// TIA Portal V21 export
DATA_BLOCK "SET VALUE"   // DB85
{ S7_Optimized_Access := 'FALSE' }
   VAR
      "PWD DOSING TIME" : String[80] := '  DOSING TIME (SEC)          :      60      ';
      "PWD WTR INLET TIME" : String[80] := '  WATER INLET TIME (MIN)     :       7     ';
      "PWD CRC TIME" : String[80] := '  CIRCULATION TIME (MIN)     :      10   ';
      "PWD DRAIN TIME" : String[80] := '  DRAIN TIME (MIN)           :       7    ';
      "STERILE TEMP1" : String[80] := '  HEAT UP-1 (DEG.C)          :    105.0  ';
      "STERILE TEMP2" : String[80] := '  HEAT UP-2 (DEG.C)          :    110.0  ';
      "STERILE TEMP3" : String[80] := '  HEAT UP-3 (DEG.C)          :    115.0  ';
      "STERILE TEMP4" : String[80] := '  STERILE TEMP (DEG.C)       :    121.4 ';
      "STERILE HOLD1" : String[80] := '  PULSE                      :       5    ';
      "STERILE HOLD2" : String[80] := '  PULSE                      :       5    ';
      "STERILE HOLD3" : String[80] := '  PULSE                      :       5    ';
      "STERILE HOLD4" : String[80] := '  HOLD TIME (MIN)            :      30    ';
      "WFI DSG TIME" : String[80] := '  DOSING TIME (SEC)          :      60 ';
      "WFI WTR TIME" : String[80] := '  WATER INLET TIME (MIN)     :       7 ';
      "WFI CRC TIME" : String[80] := '  CIRCULATION TIME (MIN)     :      10  ';
      "WFI DRAIN TIME" : String[80] := '  DRAIN TIME (MIN)           :      10  ';
      "STERILE EXH PRESS" : String[80] := '  EXHAUST PRESSURE (BAR)     :     0.05';
      "DRY VCC" : String[80] := '  VACUUM (BAR)               :    -0.500';
      "DRY VCC TIME" : String[80] := '  HOLD TIME (MIN)            :            ';
      "DRY ATS PRESSURE" : String[80] := '  ATMOSPHERIC PRESSURE (BAR) :    -0.050';
      "DRY TIME" : String[80] := '  DRYING TIME(MIN)           :      20     ';
      "PWD TEMP" : String[80] := '  PWD TEMP (DEG.C)           :     0.0    ';
      "STD TEMP1" : String[80] := '  HEAT UP-1 TEMPERATURE (DEG.C)         :   114.0       ';
      "STD TEMP2" : String[80] := '  HEAT UP-2 TEMPERATURE (DEG.C)         :   116.0       ';
      "STD TEMP3" : String[80] := '  HEAT UP-3 TEMPERATURE (DEG.C)         :   119.0       ';
      "STD TIME1" : String[80] := '  HEAT UP-1 HOLD TIME (MIN)             :      5     ';
      "STD TIME2" : String[80] := '  HEAT UP-2 HOLD TIME (MIN)             :      3     ';
      "STD TIME3" : String[80] := '  HEAT UP-3 HOLD TIME (MIN)             :      2     ';
      LEAK : String[80] := '  VACUUM (BAR)               :    -0.700';
      "DELAY BEFORE HOLD" : String[80] := '  DELAY BEFORE HOLD (MIN)    :       5';
      ACCEPTANCE : String[80] := '  ACCEPTANCE LEAKAGE (BAR)   :     0.013';
      "VCC HOLD" : String[80] := '  HOLD TIME (MIN)            :     10     ';
      "VCC PRESS" : String[80] := '  VENT PRESSURE (BAR)        :    -0.08';
      "HPHV VCC" : String[80] := '  PRE-VACUUM LEVEL (BAR)                :   -0.700      ';
      "HPHV VCC HOLD" : String[80] := '  PRE-VACUUM HOLD TIME (MIN)            :      3        ';
      "HPHV HEATUP" : String[80] := '  STERILIZATION TEMPERATURE (DEG.C)     :   121.4        ';
      "HPHV HEATUP HOLD" : String[80] := '  STERILIZATION HOLD TIME (MIN)         :     30       ';
      "HPHV NO" : String[80] := '  PRE-PULSE NUMBER                      :      3        ';
      "HPHV ATS" : String[80] := '  POST-VACUUM LEVEL (BAR)               :   -0.700      ';
      "HPHV ATS HOLD" : String[80] := '  POST-VACUUM HOLD TIME (MIN)           :     15        ';
      "HPHV EXH PRESS" : String[80] := '  EXHAUST PRESSURE (BAR)                :    0.2         ';
      "HPHV HEATUP PRESS" : String[80] := '  PRE-HEAT PRESSURE (BAR)               :    0.7        ';
      "HPHV END PRESS" : String[80] := '  END PRESSURE (BAR)                    :   -0.08       ';
      "BOW VCC" : String[80] := '  PRE-VACUUM LEVEL (BAR)                :   -0.700      ';
      "BOW VCC HOLD" : String[80] := '  PRE-VACUUM HOLD TIME (MIN)            :      3        ';
      "BOW HEATUP" : String[80] := '  STERILIZATION TEMPERATURE (DEG.C)     :   121.4        ';
      "BOW HEATUP HOLD" : String[80] := '  STERILIZATION HOLD TIME (MIN)         :     10       ';
      "BOW PRE PULSES" : String[80] := '  PRE-PULSE NUMBER                      :      3        ';
      "BOW POST VACUUM" : String[80] := '  POST-VACUUM LEVEL (BAR)               :    0.0        ';
      "BOW POST VACUUM HOLD" : String[80] := '  POST-VACUUM HOLD TIME (MIN)           :      0        ';   // 40:
      "BOW EXH PRESS" : String[80] := '  EXHAUST PRESSURE (BAR)                :    0.90        ';
      "BOW HEATUP PRESS" : String[80] := '  PRE-HEAT PRESSURE (BAR)               :    0.7        ';
      "BOW END PRESS" : String[80] := '  END PRESSURE (BAR)                    :    0.00       ';
      "STD UP PRESS" : String[80] := '  PRE PRESSURE (BAR)         :               0.00';
      "STD STOP TEMP" : String[80] := '  STERILIZATION STOP TEMP (DEG.C)       :   120.9     ';
      "STD VCC HOLD" : String[80] := '  VACUUM HOLD TIME (MIN)     :             ';
      "STD NO OF PULSES" : String[80] := '  NO OF PULSES               :                 0';
      "DONE BY" : String[80] := '';
      "DATE" : String[80] := '';
      SUMARY : String[80] := '';
      "VACUUM START" : String[80] := '';
      "VACCUM END" : String[80] := '';
      "ACTUAL LEAK" : String[80] := '';
      "ACCEPT LEAK" : String[80] := '';
      RESULT : String[80] := '';
      "PW NO OF PULSES_1" : String[80] := '$L$RNO OF PULSES               :       2         ';
      "OVERSHOOT TEMP" : String[80] := '$L$ROVERSHOOT TEMP (DEG.C)                :   124.0      ';
      "ABORT TEMP" : String[80] := '$L$RCRITICAL TEMP (DEG.C)                 :   120.5          ';
      "ABORT DELAY" : String[80] := '$L$RABORT DELAY (SEC)          :       1       ';
      "SET WFI COUNTS" : String[80] := '$L$RNO OF PULSES               :       0        ';
      "SET HPHV HT1" : String[80] := '  HEAT UP-1 TEMPEARUTRE (DEG.C)         :   114.0       ';
      "SET HPHV HT2" : String[80] := '  HEAT UP-2 TEMPEARUTRE (DEG.C)         :   116.0       ';
      "SET HPHV HT3" : String[80] := '  HEAT UP-3 TEMPEARUTRE (DEG.C)         :   119.0        ';
      "SET HPHV UP T1" : String[80] := '  HEAT UP-1 HOLD TIME (MIN)             :      5     ';
      "SET HPHV UP T2" : String[80] := '  HEAT UP-2 HOLD TIME (MIN)             :      3     ';
      "SET HPHV UP T3" : String[80] := '  HEAT UP-3 HOLD TIME (MIN)             :      2     ';
      "SET BOW HT1" : String[80] := '  HEAT UP-1 TEMPEARUTRE (DEG.C)         :   114.0     ';
      "SET BOW HT2" : String[80] := '  HEAT UP-2 TEMPEARUTRE (DEG.C)         :   116.0      ';
      "SET BOW HT3" : String[80] := '  HEAT UP-3 TEMPEARUTRE (DEG.C)         :   119.0      ';
      "SET BOW UP T1" : String[80] := '  HEAT UP-1 HOLD TIME (MIN)             :      5     ';
      "SET BOW UP T2" : String[80] := '  HEAT UP-2 HOLD TIME (MIN)             :      3     ';
      "SET BOW UP T3" : String[80] := '  HEAT UP-3 HOLD TIME (MIN)             :      2     ';
      "SET HPHV POST PULSES" : String[80] := '  POST-PULSE NUMBER                     :      1        ';
      "SET BOW POST PULSES" : String[80] := '  POST-PULSE NUMBER                     :      0        ';
      "SET BOW STOP TMP" : String[80] := '  STERILIZATION STOP TEMP (DEG.C)       :   120.9     ';   // :41
      "SET HPHV STOP TMP" : String[80] := '  STERILIZATION STOP TEMP (DEG.C)       :   120.9     ';
      "CONTROL BAND" : String[80] := '  CONTROL BAND TEMP (DEG.C)             :     0.2         ';
      "JACKET ALM TIME" : String[80] := '  JACKET ALARM TIME (MIN)               :     10                   ';
      "HEAT ALM TIME" : String[80] := '  HEATUP ALARM TIME (MIN)               :     10                   ';
      "PRINT INTERVAL" : String[80] := '  PRINT INTERVAL TIME (SEC)             :     60               ';
      "STD STERILE TEMP" : String[80] := '  STERILIZATION TEMPERATURE (DEG.C)     :   121.4        ';
      "STD STERILE HOLD" : String[80] := '  STERILIZATION HOLD TIME (MIN)         :     10       ';
      "STD END PRESSURE" : String[80] := '  END PRESSURE (BAR)                    :    0.08       ';
      AMP_LEAK : String[80] := '  VACUUM (BAR)               :    -0.700';
      "AMPVCC HOLD" : String[80] := '  HOLD TIME (MIN)            :     10     ';
      "AMP VCC PRESS" : String[80] := '  VENT PRESSURE (BAR)        :    -0.08';
   END_VAR
BEGIN
END_DATA_BLOCK
